FUNCTION_BLOCK FB_Auto_PC
VAR_INPUT
	bEnable				: BOOL;
END_VAR	
VAR_OUTPUT
	fPCV				: LREAL;
	fSCV				: LREAL;

END_VAR
VAR
	//Valvesignals
fPCV_startpos				: LREAL;
fPCV_sine					: LREAL;
fPCV_Off					: LREAL;

fSCV_On						: LREAL;
fSCV_Off					: LREAL;

	//Function Blocks
	fbAutoStartPos		: FB_AutoStartPos;
	fbAutoSineMotion	: FB_AutoSineMotion;
	
	fbClock				: FB_Clock;
	fbMUX_selector		: FB_MUX_selector;
	
	
	bStartPosOK			: BOOL;

END_VAR
VAR // added by the converter: edge detectors and wires of the graphical bodies
    _w1 : LREAL;
    _w2 : BOOL;
END_VAR

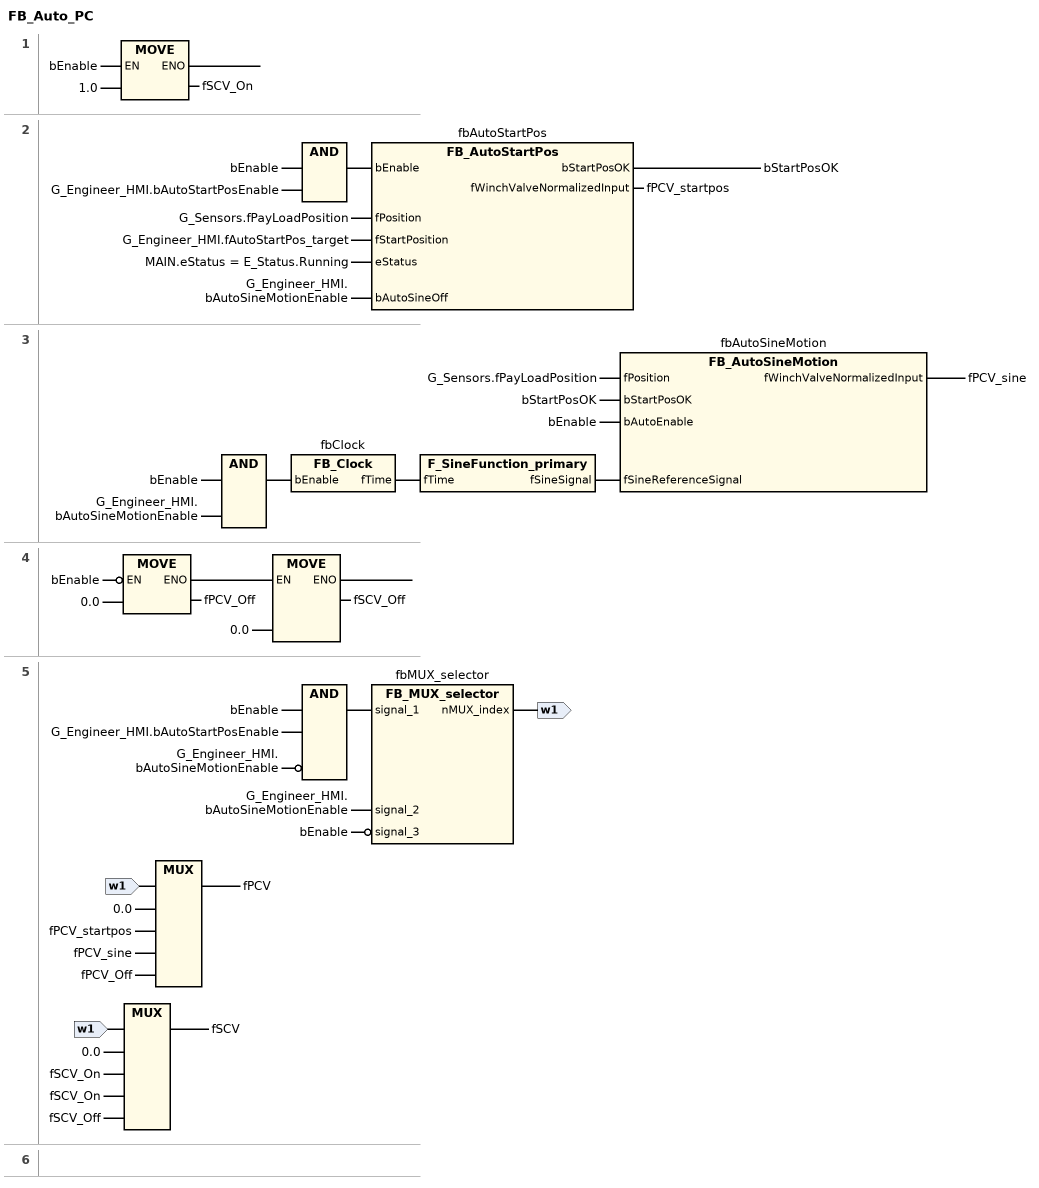
// NETWORK 1
IF bEnable THEN fSCV_On := 1.0; END_IF

// NETWORK 2
fbAutoStartPos(
    bEnable := bEnable AND G_Engineer_HMI.bAutoStartPosEnable,
    fPosition := G_Sensors.fPayLoadPosition,
    fStartPosition := G_Engineer_HMI.fAutoStartPos_target,
    eStatus := MAIN.eStatus = E_Status.Running,
    bAutoSineOff := G_Engineer_HMI.bAutoSineMotionEnable,
    fWinchValveNormalizedInput => fPCV_startpos); // FB_AutoStartPos
bStartPosOK := fbAutoStartPos.bStartPosOK;

// NETWORK 3
fbClock(bEnable := bEnable AND G_Engineer_HMI.bAutoSineMotionEnable); // FB_Clock
F_SineFunction_primary(fTime := fbClock.fTime, fSineSignal => _w1);
fbAutoSineMotion(
    fPosition := G_Sensors.fPayLoadPosition,
    bStartPosOK := bStartPosOK,
    bAutoEnable := bEnable,
    fSineReferenceSignal := _w1); // FB_AutoSineMotion
fPCV_sine := fbAutoSineMotion.fWinchValveNormalizedInput;

// NETWORK 4
_w2 := NOT bEnable;
IF _w2 THEN fPCV_Off := 0.0; END_IF
IF _w2 THEN fSCV_Off := 0.0; END_IF

// NETWORK 5
fbMUX_selector(
    signal_1 := bEnable AND G_Engineer_HMI.bAutoStartPosEnable AND NOT G_Engineer_HMI.bAutoSineMotionEnable,
    signal_2 := G_Engineer_HMI.bAutoSineMotionEnable,
    signal_3 := NOT bEnable); // FB_MUX_selector
fPCV := MUX(fbMUX_selector.nMUX_index, 0.0, fPCV_startpos, fPCV_sine, fPCV_Off);
fSCV := MUX(fbMUX_selector.nMUX_index, 0.0, fSCV_On, fSCV_On, fSCV_Off);

// NETWORK 6

END_FUNCTION_BLOCK

(* stored: Version 1.1.0.1
   POU FB_Auto_PC: Id {08676a61-e483-474a-90df-258b50adcd27}, SpecialFunc None *)
